FUNCTION_BLOCK FB_BaseExecutiveElement_HMI EXTENDS FB_BaseComponent_HMI IMPLEMENTS ITF_BaseExecutiveElement_HMI
VAR
	itfBaseExecutiveElementConnector	: ITF_BaseExecutiveElement_HMI_Connector;
	refstBaseExecutiveElementDataHMI	: REFERENCE TO ST_BaseExecutiveElement_HMI;
END_VAR

END_FUNCTION_BLOCK

(* stored: Version 1.1.0.1
   POU FB_BaseExecutiveElement_HMI: Id {f7e14e4d-7841-0cfb-1cf8-aac3b29affb7}, SpecialFunc None *)
